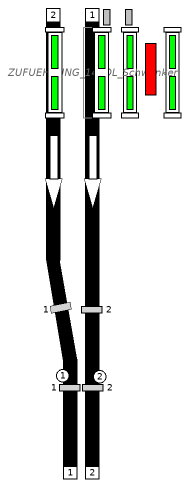
embedded screen at (73,127)-(90,200): SIGNS_ARROWDOWN
rounded rectangle at (74,0)-(88,14): text "1"; alarm colour if ST03_562_B69_0.BitInToCheck; tooltip ST03_562_B69_0
rounded rectangle at (74,458)-(88,471): text "2"; alarm colour if ST03_563_B70_7.BitInToCheck; tooltip ST03_563_B70_7
ellipse at (82,362)-(95,375): text "2"; alarm colour if ST03_563_B70_6.BitInToCheck; tooltip ST03_563_B70_6
rectangle at (71,376)-(92,383): alarm colour if ST03_563_B70_4.ValveSensor; tooltip ST03_563_B70_3
rectangle at (36,373)-(49,386): text "1"
rectangle at (92,373)-(105,386): text "2"
embedded screen at (110,19)-(170,110): ZUFUEHRUNG_268POL_RP_SCHWENKER; invisible if NOT ST03_564_Y71_5.SensorInitIn[1].SensorSignal
rectangle at (114,1)-(121,17): alarm colour if ST03_564_Y71_5.SensorInitIn[1].SensorSignal; tooltip ST03_564_Y71_5.SensorInitIn[1].SensorSignal
rectangle at (92,1)-(99,17): alarm colour if ST03_564_Y71_5.SensorWorkIn[1].SensorSignal; tooltip ST03_564_Y71_5.SensorWorkIn[1].SensorSignal
embedded screen at (72,19)-(91,110): ZUFUEHRUNG_14POL_Schwenker; invisible if NOT ST03_512_B69_6.ValveSensor
rectangle at (48,376)-(69,383): alarm colour if ST03_562_B69_4.ValveSensor; tooltip ST03_564_Y71_1
rounded rectangle at (52,458)-(66,471): text "1"; alarm colour if ST03_562_B67_7.BitInToCheck; tooltip ST03_562_B67_7
ellipse at (45,361)-(58,374): text "1"; alarm colour if ST03_562_B69_6.BitInToCheck; tooltip ST03_562_B69_6
embedded screen at (34,19)-(100,110): ZUFUEHRUNG_268POL_RP_SCHWENKER; invisible if NOT ST03_564_Y71_5.SensorWorkIn[1].SensorSignal
embedded screen at (34,127)-(51,200): SIGNS_ARROWDOWN
rectangle at (70,298)-(91,305): alarm colour if ST03_563_B70_2.ValveSensor; tooltip ST03_564_Y71_2
rectangle at (28,295)-(41,308): text "1"
rectangle at (91,295)-(104,308): text "2"
polygon at (39,294)-(60,305): alarm colour if ST03_562_B69_2.ValveSensor; tooltip ST03_564_Y71_0
rounded rectangle at (134,35)-(145,87): alarm colour if ST03_Init_Lockings.b_freiFuerSG; tooltip b_freiFuerSG
rounded rectangle at (35,0)-(49,14): text "2"; alarm colour if ST03_563_B70_0.BitInToCheck; tooltip ST03_563_B70_0
5 more shapes without text or variables
*)

(* Visualisation ZUFUEHRUNG_268POL_RP_SCHWENKER
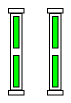
rectangle at (44,8)-(50,40): invisible if NOT $Reihe1$
rectangle at (44,47)-(50,79): invisible if NOT $Reihe1$
rounded rectangle at (39,0)-(55,5): invisible if NOT ST03_564_Y71_5.SensorWorkIn[1].SensorSignal; alarm colour if $Reihe1$; tooltip ST03_565_B72_0
rounded rectangle at (39,82)-(55,87): invisible if NOT ST03_564_Y71_5.SensorWorkIn[1].SensorSignal; alarm colour if $Reihe1$; tooltip ST03_565_B72_0
rectangle at (5,8)-(11,40): invisible if NOT $Reihe2$
rectangle at (5,47)-(11,79): invisible if NOT $Reihe2$
rounded rectangle at (0,0)-(16,5): invisible if NOT ST03_564_Y71_5.SensorWorkIn[1].SensorSignal; alarm colour if $Reihe2$; tooltip ST03_565_B72_1
rounded rectangle at (0,82)-(16,87): invisible if NOT ST03_564_Y71_5.SensorWorkIn[1].SensorSignal; alarm colour if $Reihe2$; tooltip ST03_565_B72_1
2 more shapes without text or variables
*)

(* Visualisation ZUFUEHRUNG_33POL
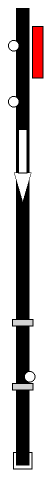
embedded screen at (9,126)-(26,199): SIGNS_ARROWDOWN
ellipse at (3,37)-(14,48): alarm colour if ST03_571_B69_0.BitInToCheck; tooltip ST03_501_B69_0
ellipse at (19,368)-(30,379): alarm colour if ST03_571_B69_6.BitInToCheck; tooltip ST03_501_B69_6
rectangle at (7,380)-(28,387): alarm colour if ST03_571_B69_5.ValveSensor; tooltip ST03_501_B69_3
rectangle at (7,316)-(28,323): alarm colour if ST03_571_B69_3.ValveSensor; tooltip ST03_501_B69_1
rounded rectangle at (8,449)-(27,466): alarm colour if ST03_571_B69_7.BitInToCheck; tooltip ST03_502_B70_0
rounded rectangle at (27,23)-(38,75): alarm colour if ST03_Init_Lockings.b_freiFuerSG; tooltip b_freiFuerSG
ellipse at (3,93)-(14,104): alarm colour if ST03_571_B69_1.BitInToCheck; tooltip ST03_501_B69_0
2 more shapes without text or variables
*)

(* Visualisation ZUFUEHRUNG_35POL
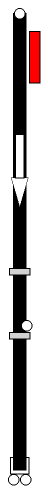
ellipse at (6,466)-(17,477): alarm colour if ST08_412_B58_6_35pol.BitInToCheck; tooltip ST08_412_B58_6_35pol
embedded screen at (9,126)-(26,199): SIGNS_ARROWDOWN
ellipse at (18,466)-(29,477): alarm colour if ST08_412_B58_5_35pol.BitInToCheck; tooltip ST08_412_B58_5_35pol
ellipse at (12,0)-(23,11): alarm colour if ST08_412_B58_4.BitInToCheck; tooltip ST08_412_B58_4
ellipse at (19,312)-(30,323): alarm colour if ST08_412_B58_7.BitInToCheck; tooltip ST08_412_B58_7
rectangle at (7,324)-(28,331): alarm colour if ST08_412_B58_2.ValveSensor; tooltip ST08_412_B58_2
rectangle at (7,260)-(28,267): alarm colour if ST08_412_B58_0.ValveSensor; tooltip ST08_412_B58_0
rounded rectangle at (8,449)-(27,466): alarm colour if ST08_412_B59_0.BitInToCheck; tooltip ST08_412_B59_0
rounded rectangle at (27,23)-(38,75): alarm colour if ST03_Init_Lockings.b_freiFuerSG; tooltip b_freiFuerSG
2 more shapes without text or variables
*)

(* Visualisation ZUFUEHRUNG_46POL
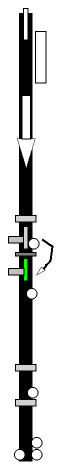
ellipse at (37,446)-(48,457): alarm colour if ST03_462_B70_1.BitInToCheck; tooltip ST03_462_B70_1
embedded screen at (23,92)-(41,165): SIGNS_ARROWDOWN
ellipse at (20,446)-(31,457): alarm colour if ST03_462_B70_2.BitInToCheck; tooltip ST03_462_B70_2
ellipse at (37,434)-(48,445): alarm colour if ST03_463_B70_7.BitInToCheck; tooltip ST03_463_B70_7
ellipse at (33,384)-(44,395): alarm colour if ST03_461_B69_7.BitInToCheck; tooltip ST03_461_B69_7
rectangle at (21,396)-(42,403): alarm colour if ST03_461_B69_2.ValveSensor; tooltip ST03_461_B69_2
rectangle at (21,361)-(42,368): alarm colour if ST03_461_B69_0.ValveSensor; tooltip ST03_461_B69_0
rounded rectangle at (41,28)-(52,80): alarm colour if ST03_Init_Lockings.b_freiFuerSG; tooltip b_freiFuerSG
rounded rectangle at (29,5)-(34,37): alarm colour if ST03_461_B69_4.BitInToCheck; tooltip ST03_461_B69_4
rectangle at (21,212)-(42,219): alarm colour if ST03_461_B69_5.ValveSensor; tooltip ST03_461_B69_5
rectangle at (14,233)-(30,240): invisible if NOT ST03_463_B70_5.ValveSensor; alarm colour if ST03_464_B71_6.BitInToCheck; tooltip ST03_464_B71_6; x offset ST03_CallFBs.ST03_463_B70_3_4_pos
rectangle at (29,223)-(34,246): invisible if NOT ST03_463_B70_5.ValveSensor; alarm colour if ST03_462_B70_0.BitInToCheck
rectangle at (29,255)-(34,278): invisible if NOT ST03_463_B70_6.ValveSensor
rectangle at (14,265)-(30,272): invisible if NOT ST03_463_B70_6.ValveSensor; alarm colour if ST03_464_B71_6.BitInToCheck; tooltip ST03_464_B71_6; x offset ST03_CallFBs.ST03_463_B70_3_4_pos
ellipse at (32,285)-(43,296): alarm colour if ST03_464_B71_7.BitInToCheck; tooltip ST03_464_B71_7
curve at (48,236)-(58,266): invisible if NOT ST03_463_B70_5.ValveSensor AND NOT NOT ST03_463_B70_5.ValveSensor
polygon at (42,264)-(51,272): invisible if NOT ST03_463_B70_5.ValveSensor AND NOT NOT ST03_463_B70_5.ValveSensor
ellipse at (34,235)-(45,246): alarm colour if ST03_462_B70_0.BitInToCheck; tooltip ST03_462_B70_0
2 more shapes without text or variables
*)

(* Visualisation ZUFUEHRUNG_48POL
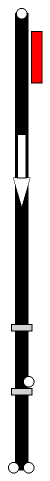
embedded screen at (9,126)-(26,199): SIGNS_ARROWDOWN
ellipse at (12,0)-(23,11): alarm colour if ST03_551_B69_0.BitInToCheck; tooltip ST03_541_B69_0
ellipse at (19,368)-(30,379): alarm colour if ST03_551_B69_6.BitInToCheck; tooltip ST03_541_B69_6
rectangle at (7,380)-(28,387): alarm colour if ST03_551_B69_4.ValveSensor; tooltip ST03_541_B69_3
rectangle at (7,316)-(28,323): alarm colour if ST03_551_B69_2.ValveSensor; tooltip ST03_541_B69_1
rounded rectangle at (27,23)-(38,75): alarm colour if ST03_Init_Lockings.b_freiFuerSG; tooltip b_freiFuerSG
ellipse at (4,454)-(15,465): alarm colour if ST03_552_B70_0.BitInToCheck; tooltip ST03_542_B70_0
ellipse at (19,454)-(30,465): alarm colour if ST03_551_B69_7.BitInToCheck; tooltip ST03_542_B70_0
2 more shapes without text or variables
*)

(* Visualisation ZUFUEHRUNG_72POL
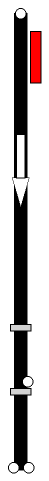
embedded screen at (9,126)-(26,199): SIGNS_ARROWDOWN
ellipse at (12,0)-(23,11): alarm colour if ST03_546_B69_0.BitInToCheck; tooltip ST03_541_B69_0
ellipse at (19,368)-(30,379): alarm colour if ST03_546_B69_6.BitInToCheck; tooltip ST03_541_B69_6
rectangle at (7,380)-(28,387): alarm colour if ST03_546_B69_4.ValveSensor; tooltip ST03_541_B69_3
rectangle at (7,316)-(28,323): alarm colour if ST03_546_B69_2.ValveSensor; tooltip ST03_541_B69_1
rounded rectangle at (27,23)-(38,75): alarm colour if ST03_Init_Lockings.b_freiFuerSG; tooltip b_freiFuerSG
ellipse at (5,454)-(16,465): alarm colour if ST03_547_B70_0.BitInToCheck; tooltip ST03_542_B70_0
ellipse at (20,454)-(31,465): alarm colour if ST03_546_B69_7.BitInToCheck; tooltip ST03_542_B70_0
2 more shapes without text or variables
*)

(* Visualisation ZUFUEHRUNG_74_91_168POL
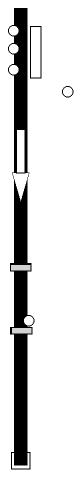
rounded rectangle at (8,444)-(27,461): invisible if NOT MP.ST03.SGM_3621; alarm colour if ST03_422_B64_4.BitInToCheck
ellipse at (5,35)-(16,46): invisible if MP.ST03.SGM_3621; alarm colour if ST08_412_B58_5.BitInToCheck
embedded screen at (9,121)-(26,194): SIGNS_ARROWDOWN
ellipse at (5,56)-(16,67): invisible if MP.ST03.SGM_3621 OR gTypeCode=379; alarm colour if ST08_412_B58_6.BitInToCheck
ellipse at (5,17)-(16,28): invisible if MP.ST03.SGM_3621; alarm colour if ST08_412_B58_4.BitInToCheck
ellipse at (19,307)-(30,318): invisible if MP.ST03.SGM_3621; alarm colour if ST08_412_B58_7.BitInToCheck
rectangle at (7,319)-(28,326): invisible if MP.ST03.SGM_3621; alarm colour if ST08_412_B58_2.ValveSensor
rectangle at (7,255)-(28,262): invisible if MP.ST03.SGM_3621; alarm colour if ST08_412_B58_0.ValveSensor
rounded rectangle at (8,444)-(27,461): invisible if MP.ST03.SGM_3621; alarm colour if ST08_412_B59_0.BitInToCheck; tooltip ST08_412_B59_0
rounded rectangle at (27,18)-(38,70): alarm colour if ST03_Init_Lockings.b_freiFuerSG; tooltip b_freiFuerSG
rectangle at (8,319)-(29,326): invisible if NOT MP.ST03.SGM_3621; alarm colour if ST03_421_B63_2.ValveSensor; tooltip ST03_421_B63_2
ellipse at (5,35)-(16,46): invisible if NOT MP.ST03.SGM_3621; alarm colour if ST03_421_B63_5.BitInToCheck; tooltip ST03_421_B63_5
ellipse at (59,78)-(70,89): invisible if NOT MP.ST03.SGM_3621; alarm colour if ST03_421_B63_6.BitInToCheck; tooltip ST03_421_B63_6
ellipse at (5,17)-(16,28): invisible if NOT MP.ST03.SGM_3621; alarm colour if ST03_421_B63_4.BitInToCheck; tooltip ST03_421_B63_4
rectangle at (7,256)-(28,263): invisible if NOT MP.ST03.SGM_3621; alarm colour if ST03_421_B63_0.ValveSensor; tooltip ST03_421_B63_0
ellipse at (20,307)-(31,318): invisible if NOT MP.ST03.SGM_3621; alarm colour if ST03_421_B63_7.BitInToCheck; tooltip ST03_421_B63_7
2 more shapes without text or variables
*)

(* Visualisation ZUFUEHRUNG_7POL
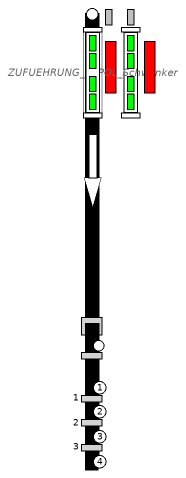
embedded screen at (16,126)-(33,199): SIGNS_ARROWDOWN
ellipse at (18,0)-(30,12): alarm colour if ST03_514_B71_7.BitInToCheck; tooltip ST03_514_B71_7
ellipse at (25,332)-(36,343): alarm colour if ST03_513_B70_4.BitInToCheck; tooltip ST03_513_B70_4
rectangle at (13,344)-(34,351): alarm colour if ST03_513_B70_3. ValveSensor; tooltip ST03_513_B70_3
rectangle at (13,309)-(34,327): alarm colour if ST03_513_B70_0.ValveSensor; tooltip ST03_513_B70_0
rounded rectangle at (37,33)-(48,85): alarm colour if ST03_Init_Lockings.b_freiFuerSG; tooltip b_freiFuerSG
ellipse at (25,447)-(38,460): text "4"; alarm colour if ST03_514_B71_6.BitInToCheck; tooltip ST03_514_B71_6
ellipse at (25,422)-(38,435): text "3"; alarm colour if ST03_514_B71_5.BitInToCheck; tooltip ST03_514_B71_5
rectangle at (13,436)-(34,443): alarm colour if ST03_514_B71_4.ValveSensor; tooltip ST03_514_B71_4
ellipse at (25,397)-(38,410): text "2"; alarm colour if ST03_514_B71_2.BitInToCheck; tooltip ST03_514_B71_2
rectangle at (13,411)-(34,418): alarm colour if ST03_514_B71_1.ValveSensor; tooltip ST03_514_B71_1
ellipse at (25,373)-(38,386): text "1"; alarm colour if ST03_513_B70_7.BitInToCheck; tooltip ST03_513_B70_7
rectangle at (13,387)-(34,394): alarm colour if ST03_513_B70_6.ValveSensor; tooltip ST03_513_B70_6
rectangle at (1,383)-(14,396): text "1"
rectangle at (1,408)-(14,421): text "2"
rectangle at (1,432)-(14,445): text "3"
embedded screen at (53,19)-(72,110): ZUFUEHRUNG_7POL_Schwenker; invisible if NOT ST03_515_Y72_1.SensorInitIn[1].SensorSignal
rectangle at (59,1)-(66,17): alarm colour if ST03_515_Y72_1.SensorInitIn[1].SensorSignal; tooltip ST03_515_Y72_1
rectangle at (37,1)-(44,17): alarm colour if ST03_515_Y72_1.SensorWorkIn[1].SensorSignal; tooltip ST03_515_Y72_1
embedded screen at (15,19)-(34,110): ZUFUEHRUNG_14POL_Schwenker; invisible if NOT ST03_512_B69_6.ValveSensor
embedded screen at (15,19)-(34,110): ZUFUEHRUNG_7POL_Schwenker; invisible if NOT ST03_515_Y72_1.SensorWorkIn[1].SensorSignal
rounded rectangle at (76,33)-(87,85): alarm colour if ST00_73_K4.BitInToCheck; tooltip ST00_73_K4
3 more shapes without text or variables
*)

(* Visualisation ZUFUEHRUNG_7POL_SCHWENKER
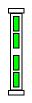
rectangle at (5,8)-(11,23): invisible if NOT ST03_512_XG1.BitInToCheck
rectangle at (5,25)-(11,40): invisible if NOT ST03_512_XG1.BitInToCheck
rectangle at (5,47)-(11,62): invisible if NOT ST03_512_XG1.BitInToCheck
rectangle at (5,64)-(11,79): invisible if NOT ST03_512_XG1.BitInToCheck
rounded rectangle at (0,0)-(16,5): invisible if ST03_515_Y72_1.SensorWorkIn[1].SensorSignal; alarm colour if ST03_512_XG1.BitInToCheck
rounded rectangle at (0,82)-(16,87): invisible if ST03_515_Y72_1.SensorWorkIn[1].SensorSignal; alarm colour if ST03_512_XG1.BitInToCheck
1 more shapes without text or variables
*)

(* Visualisation ZUFUEHRUNG_88POL
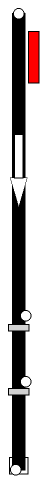
embedded screen at (9,126)-(26,199): SIGNS_ARROWDOWN
ellipse at (12,0)-(23,11): alarm colour if ST03_501_B69_0.BitInToCheck; tooltip ST03_501_B69_0
ellipse at (19,368)-(30,379): alarm colour if ST03_501_B69_6.BitInToCheck; tooltip ST03_501_B69_6
rectangle at (7,380)-(28,387): alarm colour if ST03_501_B69_3.ValveSensor; tooltip ST03_501_B69_3
rectangle at (7,316)-(28,323): alarm colour if ST03_501_B69_1.ValveSensor; tooltip ST03_501_B69_1
rounded rectangle at (8,449)-(27,466): alarm colour if ST03_502_B70_0.BitInToCheck; tooltip ST03_502_B70_0
rounded rectangle at (27,23)-(38,75): alarm colour if ST03_Init_Lockings.b_freiFuerSG; tooltip b_freiFuerSG
ellipse at (19,302)-(30,313): alarm colour if ST03_501_B69_5.BitInToCheck; tooltip ST03_501_B69_5
ellipse at (9,456)-(20,467): alarm colour if ST03_501_B69_7.BitInToCheck; tooltip ST03_501_B69_7
2 more shapes without text or variables
*)

(* Visualisation ZUFUEHRUNG_88POL_AMG
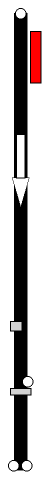
embedded screen at (9,126)-(26,199): SIGNS_ARROWDOWN
ellipse at (12,0)-(23,11): alarm colour if ST03_521_B69_0.BitInToCheck; tooltip ST03_521_B69_0
ellipse at (19,368)-(30,379): alarm colour if ST03_521_B69_6.BitInToCheck; tooltip ST03_521_B69_6
rectangle at (7,380)-(28,387): alarm colour if ST03_521_B69_4.ValveSensor; tooltip ST03_521_B69_3
rectangle at (7,313)-(19,323): alarm colour if ST03_521_B69_2.ValveSensor; tooltip ST03_521_B69_1
rounded rectangle at (27,23)-(38,75): alarm colour if ST03_Init_Lockings.b_freiFuerSG; tooltip b_freiFuerSG
ellipse at (5,452)-(16,463): alarm colour if ST03_521_B69_7.BitInToCheck; tooltip ST03_521_B69_7
ellipse at (18,452)-(29,463): alarm colour if ST03_522_B70_0.BitInToCheck; tooltip ST03_522_B70_0
2 more shapes without text or variables
*)

(* Visualisation ZUFUEHRUNG_92POL
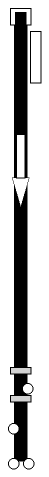
ellipse at (30,455)-(41,466): alarm colour if ST03_445_B70_1.BitInToCheck; tooltip ST03_445_B70_1
embedded screen at (19,131)-(36,204): SIGNS_ARROWDOWN
ellipse at (15,455)-(26,466): alarm colour if ST03_445_B70_2.BitInToCheck; tooltip ST03_445_B70_2
ellipse at (15,420)-(26,431): alarm colour if ST03_446_B70_4.BitInToCheck; tooltip ST03_446_B70_4
ellipse at (29,380)-(40,391): alarm colour if ST03_444_B69_7.BitInToCheck; tooltip ST03_444_B69_7
rectangle at (17,392)-(38,399): alarm colour if ST03_444_B69_2.ValveSensor; tooltip ST03_444_B69_2
rectangle at (17,364)-(38,371): alarm colour if ST03_444_B69_0.ValveSensor; tooltip ST03_444_B69_0
rounded rectangle at (17,5)-(38,22): alarm colour if ST03_435_B67_4.BitInToCheck; tooltip ST03_435_B67_4
rounded rectangle at (37,28)-(48,80): alarm colour if ST03_Init_Lockings.b_freiFuerSG; tooltip b_freiFuerSG
2 more shapes without text or variables
*)

(* Visualisation ZUFUEHRUNG_93POL
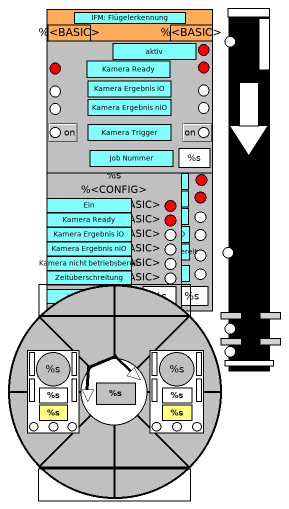
embedded screen at (40,160)-(206,303): ZLIB_SENSOPART_1; invisible if gTypeCode<>4991 AND gTypeCode <>312 OR MP.ST02.SensopartEthernet
embedded screen at (40,160)-(175,303): ZLIB_SENSOPART_5; invisible if gTypeCode<>4991 AND gTypeCode <>312 OR NOT MP.ST02.SensopartEthernet
embedded screen at (0,276)-(215,493): ROUNDTABLE; invisible if gTypeCode<>4991 AND gTypeCode <>312
embedded screen at (40,1)-(206,165): ZLIB_IFM; invisible if gTypeCode<>4991 AND gTypeCode <>312
ellipse at (218,28)-(229,39): alarm colour if NOT ST02_FDB_40_B61.BitInToCheck; tooltip ST02_FDB_40_B61
embedded screen at (223,74)-(261,147): SIGNS_ARROWDOWN
ellipse at (218,315)-(229,326): alarm colour if ST00_72_X1_3.BitInToCheck; tooltip ST00_72_X1_3
rectangle at (214,304)-(235,311): alarm colour if ST00_74_Y2_5.SensorWorkIn[1].SensorSignal; tooltip ST00_74_Y2_5
rectangle at (253,304)-(274,311): alarm colour if ST00_74_Y2_5.SensorWorkIn[2].SensorSignal; tooltip ST00_74_Y2_5
rectangle at (214,330)-(235,337): alarm colour if NOT ST00_74_Y2_4.SensorWorkIn[1].SensorSignal; tooltip ST00_74_Y2_4
rectangle at (253,330)-(274,337): alarm colour if NOT ST00_74_Y2_4.SensorWorkIn[2].SensorSignal; tooltip ST00_74_Y2_4
rectangle at (222,342)-(263,363): invisible if gTypeCode<>4991
ellipse at (218,338)-(229,349): invisible if gTypeCode<>4991; alarm colour if ST02_FDB_80_B02.BitInToCheck; tooltip ST02_FDB_80_B02
rectangle at (218,352)-(267,358): invisible if gTypeCode<>4991
ellipse at (216,239)-(227,250): alarm colour if NOT ST02_FDB_40_B71.BitInToCheck; tooltip ST02_FDB_40_B71
rectangle at (225,149)-(259,156): alarm colour if ST02_FDB_54_B41.BitInToCheck
rounded rectangle at (252,10)-(263,62): alarm colour if ST03_Init_Lockings.b_freiFuerSG; tooltip b_freiFuerSG
rounded rectangle at (221,0)-(263,9): alarm colour if ST02_S1_40K01.BitInToCheck; tooltip ST02_S1_40K01
rectangle at (222,194)-(262,200): alarm colour if ST02_FDB_54_B21.ValveSensor
1 more shapes without text or variables
*)

(* Visualisation ZUFUEHRUNG_NOX_4POL
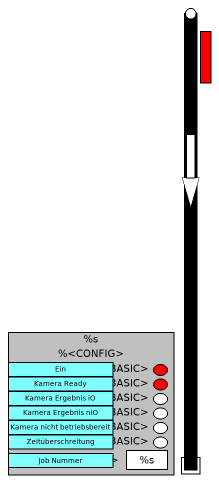
embedded screen at (174,126)-(191,199): SIGNS_ARROWDOWN
ellipse at (177,0)-(188,11): alarm colour if ST03_491_B69_0.BitInToCheck; tooltip ST03_491_B69_0
ellipse at (6,394)-(17,405): alarm colour if ST03_491_B69_5.BitInToCheck; tooltip ST03_491_B69_5
rectangle at (7,406)-(28,413): alarm colour if ST03_491_B69_2.ValveSensor; tooltip ST03_491_B69_2
rectangle at (7,371)-(28,378): alarm colour if ST03_491_B69_1.ValveSensor; tooltip ST03_491_B69_1
rounded rectangle at (173,449)-(192,466): alarm colour if ST03_491_B69_7.BitInToCheck; tooltip ST03_491_B69_7
rounded rectangle at (192,23)-(203,75): alarm colour if ST03_Init_Lockings.b_freiFuerSG; tooltip b_freiFuerSG
embedded screen at (0,324)-(166,467): ZLIB_SENSOPART_5; invisible if TRUE
2 more shapes without text or variables
*)

(* Visualisation ZUFUEHRUNG_NOX_5_6POL
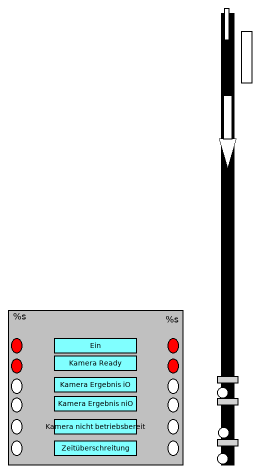
embedded screen at (274,87)-(291,160): SIGNS_ARROWDOWN
ellipse at (272,445)-(283,456): alarm colour if ST03_4x3_B70_1.BitInToCheck; tooltip ST03_4x3_B70_1
ellipse at (273,419)-(284,430): alarm colour if ST03_4x3_B70_0.BitInToCheck; tooltip ST03_4x3_B70_0
rectangle at (272,431)-(293,438): alarm colour if ST03_4x2_B69_7.ValveSensor; tooltip ST03_4x2_B69_7
rectangle at (272,390)-(293,397): alarm colour if ST03_4x2_B69_4.ValveSensor; tooltip ST03_4x2_B69_4
rounded rectangle at (296,23)-(307,75): alarm colour if ST03_Init_Lockings.b_freiFuerSG; tooltip b_freiFuerSG
rounded rectangle at (279,0)-(284,32): alarm colour if ST03_4x2_B69_0.BitInToCheck; tooltip ST03_4x2_B69_0
rounded rectangle at (272,368)-(293,375): alarm colour if ST03_4x2_B69_2.ValveSensor; tooltip ST03_4x2_B69_2
ellipse at (272,379)-(283,390): alarm colour if ST03_4x2_B69_5.BitInToCheck; tooltip ST03_4x2_B69_5
embedded screen at (63,302)-(238,457): ZLIB_SENSOPART_6; invisible if gTypeCode <> 4993
1 more shapes without text or variables
*)

(* Visualisation DOOR_LOCK
rectangle at (0,0)-(31,31): invisible if $lock$ AND NOT $visibal_open$; alarm colour if NOT $lock$
rectangle at (0,0)-(31,31): invisible if NOT $open$
*)

(* Visualisation MIN_EXIT
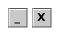
button at (1,0)-(20,19): text "_"; shows 'ST_MinExit.btn_min.Text'; invisible if ST_MinExit.btn_min.Visible; taps ST_MinExit.btn_min.Pressed; dynamic style ST_MinExit.btn_min.TextColor, ST_MinExit.btn_min.BackgroundColor, ST_MinExit.btn_min.BackgroundColor, ST_MinExit.btn_min.Enable
button at (25,0)-(44,19): text "X"; shows 'ST_MinExit.btn_exit.Text'; invisible if ST_MinExit.btn_exit.Visible; taps ST_MinExit.btn_exit.Pressed; runs INTERN EXITPROGRAM; dynamic style ST_MinExit.btn_exit.TextColor, ST_MinExit.btn_exit.BackgroundColor, ST_MinExit.btn_exit.BackgroundColor, ST_MinExit.btn_exit.Enable
*)

(* Visualisation SPRACHE_MENUE
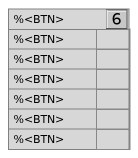
rectangle at (0,20)-(121,41): text "%<BTN>"; shows ST_Lng.btn_Language[0].Text; invisible if NOT ST_Lng.fb_ton_ausblenden.IN OR ST_Lng.btn_Language[0].unsichtbar; taps ST_Lng.btn_Language[0].tasten; runs INTERN LANGUAGE DE; dynamic style Visu.System.btn_Language[0].TextFarbe, ST_Lng.btn_Language[0].deaktivieren
rectangle at (0,40)-(121,61): text "%<BTN>"; shows ST_Lng.btn_Language[1].Text; invisible if NOT ST_Lng.fb_ton_ausblenden.IN OR ST_Lng.btn_Language[1].unsichtbar; taps ST_Lng.btn_Language[1].tasten; runs INTERN LANGUAGE EN; dynamic style Visu.System.btn_Language[1].TextFarbe, ST_Lng.btn_Language[1].deaktivieren
rectangle at (0,60)-(121,81): text "%<BTN>"; shows ST_Lng.btn_Language[2].Text; invisible if NOT ST_Lng.fb_ton_ausblenden.IN OR ST_Lng.btn_Language[2].unsichtbar; taps ST_Lng.btn_Language[2].tasten; runs INTERN LANGUAGE CZ; dynamic style Visu.System.btn_Language[2].TextFarbe, ST_Lng.btn_Language[2].deaktivieren
rectangle at (0,80)-(121,101): text "%<BTN>"; shows ST_Lng.btn_Language[3].Text; invisible if NOT ST_Lng.fb_ton_ausblenden.IN OR ST_Lng.btn_Language[3].unsichtbar; taps ST_Lng.btn_Language[3].tasten; runs INTERN LANGUAGE; dynamic style Visu.System.btn_Language[3].TextFarbe, ST_Lng.btn_Language[3].deaktivieren
rectangle at (0,100)-(121,121): text "%<BTN>"; shows ST_Lng.btn_Language[4].Text; invisible if NOT ST_Lng.fb_ton_ausblenden.IN OR ST_Lng.btn_Language[4].unsichtbar; taps ST_Lng.btn_Language[4].tasten; runs INTERN LANGUAGE; dynamic style Visu.System.btn_Language[4].TextFarbe, ST_Lng.btn_Language[4].deaktivieren
rectangle at (0,120)-(121,141): text "%<BTN>"; shows ST_Lng.btn_Language[5].Text; invisible if NOT ST_Lng.fb_ton_ausblenden.IN OR ST_Lng.btn_Language[5].unsichtbar; taps ST_Lng.btn_Language[5].tasten; runs INTERN LANGUAGE; dynamic style Visu.System.btn_Language[5].TextFarbe, ST_Lng.btn_Language[5].deaktivieren
other_BMP at (88,20)-(122,41): invisible if NOT ST_Lng.fb_ton_ausblenden.IN OR ST_Lng.btn_Language[0].unsichtbar; taps ST_Lng.btn_Language[0].tasten; dynamic style ST_Lng.btn_Language[0].BmpPath
other_BMP at (88,40)-(122,61): invisible if NOT ST_Lng.fb_ton_ausblenden.IN OR ST_Lng.btn_Language[1].unsichtbar; taps ST_Lng.btn_Language[1].tasten; dynamic style ST_Lng.btn_Language[1].BmpPath
other_BMP at (88,60)-(122,81): invisible if NOT ST_Lng.fb_ton_ausblenden.IN OR ST_Lng.btn_Language[2].unsichtbar; taps ST_Lng.btn_Language[2].tasten; dynamic style ST_Lng.btn_Language[2].BmpPath
other_BMP at (88,80)-(122,101): invisible if NOT ST_Lng.fb_ton_ausblenden.IN OR ST_Lng.btn_Language[3].unsichtbar; taps ST_Lng.btn_Language[3].tasten; dynamic style ST_Lng.btn_Language[3].BmpPath
other_BMP at (88,100)-(122,121): invisible if NOT ST_Lng.fb_ton_ausblenden.IN OR ST_Lng.btn_Language[4].unsichtbar; taps ST_Lng.btn_Language[4].tasten; dynamic style ST_Lng.btn_Language[4].BmpPath
other_BMP at (88,120)-(122,141): invisible if NOT ST_Lng.fb_ton_ausblenden.IN OR ST_Lng.btn_Language[5].unsichtbar; taps ST_Lng.btn_Language[5].tasten; dynamic style ST_Lng.btn_Language[5].BmpPath
rectangle at (0,0)-(121,21): text "%<BTN>"; shows ST_Lng.btn_Language[ST_Lng.index].Text; invisible if ST_Lng.btn_Language[ST_Lng.index].unsichtbar; taps ST_Lng.b_einblenden; dynamic style Visu.System.btn_Language[ST_System.index].TextFarbe, ST_Lng.btn_Language[ST_System.index].innenFarbe, ST_Lng.btn_Language[ST_Lng.index].deaktivieren
button at (98,1)-(119,20): text "6"; shows '0xEA'; taps ST_Lng.b_einblenden; dynamic style Color.lightgrey, Color.lightgrey
*)

(* Visualisation TEILEZAEHLER
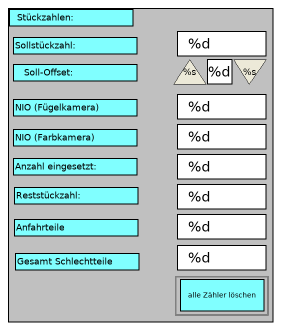
rectangle at (0,0)-(265,314): text "%<DATA>"; shows 'Parts'
rectangle at (10,23)-(157,48): text "%<DATA>"; shows 'PartsToProduce'
rectangle at (169,23)-(258,48): text "%d"; shows MP.ST00.PartsToProduce; editable 0..
rectangle at (10,51)-(157,76): text "%<DATA>"; shows 'PartsToProduceOffset'
rectangle at (199,51)-(224,76): text "%d"; shows MP.ST00.PartsToProduceOffset; editable 0..
rectangle at (10,146)-(157,171): text "%<DATA>"; shows 'gPartsInserted'
rectangle at (169,146)-(258,171): text "%d"; shows gPartsInserted; editable 0..
rectangle at (10,176)-(157,201): text "%<DATA>"; shows 'PartsRemaining'
rectangle at (169,176)-(258,201): text "%d"; shows MP.ST00.PartsRemaining; editable
embedded screen at (165,51)-(198,76): ZLIB_VISUBUTTON_ARROW_UP
embedded screen at (225,51)-(258,76): ZLIB_VISUBUTTON_ARROW_DOWN
embedded screen at (167,268)-(260,307): ZLIB_VISUBUTTON_S18
rectangle at (10,116)-(157,141): text "%<DATA>"; shows 'gNokPartsColorCam'; invisible if gTypeCode<>5633 AND gTypeCode<>4991 AND gTypeCode <>312 AND gTypeCode <>322
rectangle at (10,86)-(157,111): text "%<DATA>"; shows 'gNokPartsWingCam'; invisible if gTypeCode<>4991 AND gTypeCode <>312
rectangle at (169,86)-(258,111): text "%d"; shows gNokPartsWingCam; invisible if gTypeCode<>4991 AND gTypeCode <>312; editable 0..
rectangle at (169,116)-(258,141): text "%d"; shows gNokPartsColorCam; invisible if gTypeCode<>5633 AND gTypeCode<>4991 AND gTypeCode <>312 AND gTypeCode <>322; editable 0..
rectangle at (1,1)-(125,18): text "Stückzahlen:"; invisible if TRUE
rectangle at (5,29)-(129,46): text "Sollstückzahl:"; invisible if TRUE
rectangle at (5,56)-(129,73): text "Soll-Offset:"; invisible if TRUE
rectangle at (5,91)-(129,108): text "NIO (Fügelkamera)"; invisible if TRUE
rectangle at (5,121)-(129,138): text "NIO (Farbkamera)"; invisible if TRUE
rectangle at (5,150)-(129,167): text "Anzahl eingesetzt:"; invisible if TRUE
rectangle at (6,179)-(130,196): text "Reststückzahl:"; invisible if TRUE
rectangle at (172,271)-(256,303): text "alle Zähler löschen"; invisible if TRUE; dynamic style Color.lightgrey, Color.grey
rectangle at (10,207)-(166,232): text "%<DATA>"; shows 'Anfahrteile'
rectangle at (10,238)-(170,263): text "%<DATA>"; shows 'Gesamt Schlechtteile'
rectangle at (6,211)-(130,228): text "Anfahrteile"; invisible if TRUE
rectangle at (7,245)-(131,262): text "Gesamt Schlechtteile"; invisible if TRUE
rectangle at (169,206)-(258,231): text "%d"; shows i32_first_parts; editable 0..
rectangle at (169,237)-(258,262): text "%d"; shows i32_total_nok_parts; editable 0..
*)

(* Visualisation ZLIB_IFM
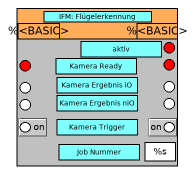
rectangle at (15,110)-(146,129): text "%<BASIC>"; shows 'Kamera Trigger'
rectangle at (15,69)-(146,88): text "%<BASIC>"; shows 'Kamera Ergebnis iO'
rectangle at (15,86)-(146,105): text "%<BASIC>"; shows 'Kamera Ergebnis niO'
ellipse at (147,73)-(158,84): alarm colour if ST02_FDB_56X1_6_IO.BitInToCheck
ellipse at (147,90)-(158,101): alarm colour if ST02_FDB_56X1_6_NIO.BitInToCheck
rectangle at (15,47)-(146,66): text "%<BASIC>"; shows 'Kamera Ready'
ellipse at (147,51)-(158,62): alarm colour if ST02_FDB_56X1_5_READY.BitInToCheck
rectangle at (40,134)-(121,153): text "%<BASIC>"; shows 'Job Nummer'
rectangle at (128,134)-(159,153): text "%s"; shows TD.IFM_CamProgNo; editable 0..3
ellipse at (147,34)-(158,45): alarm colour if MP.ST00.IFMCameraActive
ellipse at (3,74)-(14,85): alarm colour if ST02_FDB_55X1_6_IO.BitInToCheck
ellipse at (3,91)-(14,102): alarm colour if ST02_FDB_55X1_6_NIO.BitInToCheck
ellipse at (3,52)-(14,63): alarm colour if ST02_FDB_55X1_5_READY.BitInToCheck
rectangle at (62,30)-(143,49): text "%<BASIC>"; shows 'aktiv'
rectangle at (0,0)-(161,31): text "%<BASIC>"; shows 'IFM_Flügelerkennung'
rectangle at (1,15)-(43,31): text "%<BASIC>"; shows 'links'
button at (132,110)-(160,128): text "on"; invisible if ModeSelect.Mode <> 10; taps .ST02_FDB_56X1_2_TRIGGER.BitOutToSet; dynamic style color.lightgrey
ellipse at (147,114)-(158,124): alarm colour if .ST02_FDB_56X1_2_TRIGGER.BitOutToSet; taps .ST02_FDB_56X1_2_TRIGGER.BitOutToSet; dynamic style ModeSelect.Mode <> 10
button at (2,110)-(30,128): text "on"; invisible if ModeSelect.Mode <> 10; taps .ST02_FDB_55X1_2_TRIGGER.BitOutToSet; dynamic style color.lightgrey
ellipse at (3,114)-(14,124): alarm colour if .ST02_FDB_55X1_2_TRIGGER.BitOutToSet; taps .ST02_FDB_55X1_2_TRIGGER.BitOutToSet; dynamic style ModeSelect.Mode <> 10
rectangle at (64,33)-(145,49): text "aktiv"; invisible if TRUE
rectangle at (39,50)-(120,66): text "Kamera Ready"; invisible if TRUE
rectangle at (40,69)-(121,85): text "Kamera Ergebnis iO"; invisible if TRUE
rectangle at (40,87)-(121,103): text "Kamera Ergebnis niO"; invisible if TRUE
rectangle at (40,111)-(121,127): text "Kamera Trigger"; invisible if TRUE
rectangle at (42,136)-(123,152): text "Job Nummer"; invisible if TRUE
rectangle at (120,15)-(161,31): text "%<BASIC>"; shows 'rechts'
rectangle at (27,3)-(135,14): text "IFM: Flügelerkennung"; invisible if TRUE
1 more shapes without text or variables
*)

(* Visualisation ZLIB_OVERRIDE
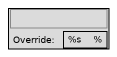
rectangle at (0,0)-(101,41): alarm colour if $override$<$overrideVorgabe$
other_SCROLLBAR at (2,1)-(99,20): top $override$; right 0; bottom 100
rounded rectangle at (0,23)-(57,41): text "Override:"; shows $override$; editable 0..100
rectangle at (55,23)-(99,40): text "%"; alarm colour if $override$<$overrideVorgabe$
rectangle at (55,23)-(99,40): text "%s"; shows $override$; editable 0..100
*)

(* Visualisation ZLIB_SCHWENKARM
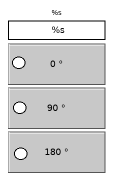
rectangle at (0,0)-(101,171): text "%s"; shows '$FB$'
rectangle at (2,13)-(99,32): text "%s"; shows $FB$.fb_state_entry.i16_step; alarm colour if $FB$.fb_state_entry.i16_step=1000
button at (2,36)-(99,77): text "0 °"; dynamic style Color.grey, TRUE
button at (2,80)-(99,121): text "90 °"; dynamic style Color.grey, TRUE
button at (2,124)-(99,165): text "180 °"; dynamic style Color.grey, TRUE
button at (2,36)-(99,77): text "0 °"; invisible if ModeSelect.Mode<>10; taps $FB$.b_0_grad; dynamic style color.lightgrey, Color.grey, ModeSelect.Mode<>10
button at (2,80)-(99,121): text "90 °"; invisible if ModeSelect.Mode<>10; taps $FB$.b_90_grad; dynamic style color.lightgrey, Color.grey, ModeSelect.Mode<>10
button at (2,124)-(99,165): text "180 °"; invisible if ModeSelect.Mode<>10; taps $FB$.b_180_grad; dynamic style color.lightgrey, Color.grey, ModeSelect.Mode<>10
ellipse at (6,49)-(19,61): alarm colour if $FB$.ST02_90_0_sens
ellipse at (7,94)-(20,106): alarm colour if $FB$.ST02_90_sens
ellipse at (8,140)-(21,152): alarm colour if $FB$.ST02_90_180_sens
*)

(* Visualisation ZLIB_ERRORHANDLER
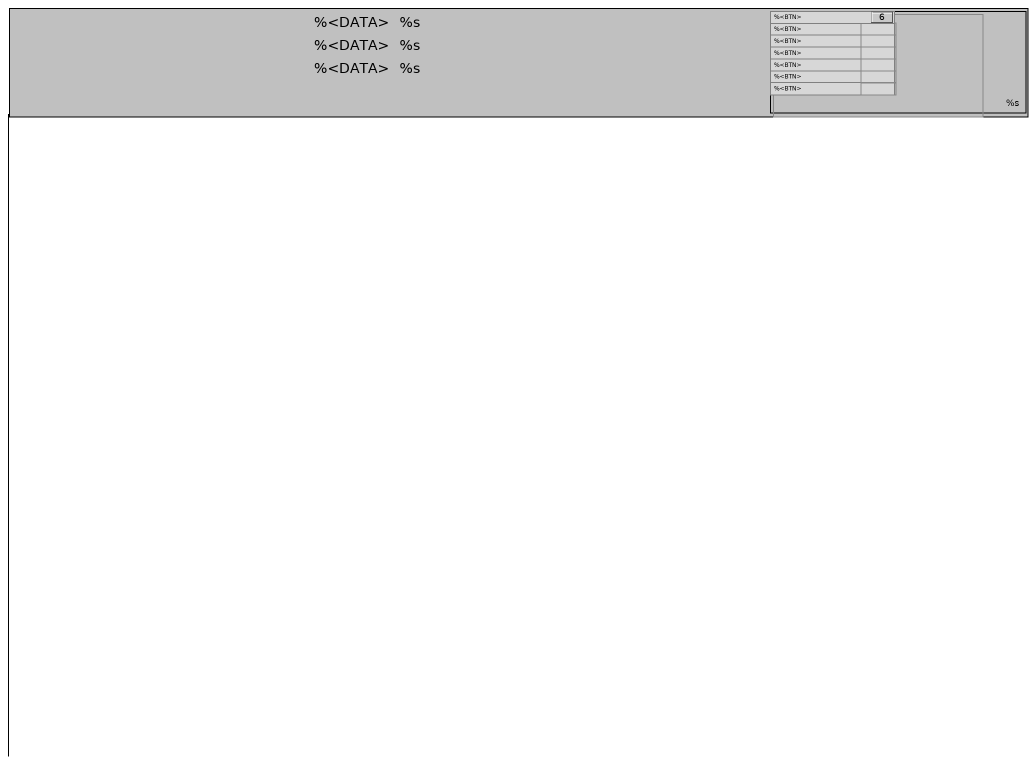
embedded screen at (0,106)-(1017,748): zLib_ErrorList
rectangle at (1,108)-(1020,759): opens ZOOMTOCALLER
rectangle at (886,87)-(1016,103): text "%s"; shows .gVarStrSystemTime
rectangle at (385,27)-(670,47): text "%s"; shows .TD.ArtNo
rectangle at (244,27)-(383,47): text "%<DATA>"; shows 'ArtNo'
rectangle at (385,4)-(670,24): text "%s"; shows .TD.TypeName
rectangle at (244,4)-(383,24): text "%<DATA>"; shows 'TypeName'
rectangle at (385,50)-(670,70): text "%s"; shows .TD.TypeDescription
rectangle at (244,50)-(383,70): text "%<DATA>"; shows 'TypeDescription'
embedded screen at (762,3)-(888,87): SPRACHE_MENUE
3 more shapes without text or variables
*)

(* Visualisation ZLIB_ERRORLINE
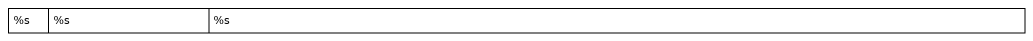
rectangle at (0,0)-(41,25): text "%s"; shows $ErrorStruct$.No; invisible if $ErrorStruct$.No = 0; dynamic style $ErrorStruct$.LineColor, $ErrorStruct$.LineColor
rectangle at (200,0)-(1017,25): text "%s"; shows $ErrorStruct$.Text; invisible if $ErrorStruct$.No = 0; dynamic style $ErrorStruct$.LineColor, $ErrorStruct$.LineColor
rectangle at (40,0)-(201,25): text "%s"; shows $ErrorStruct$.DateTime; invisible if $ErrorStruct$.No = 0; dynamic style $ErrorStruct$.LineColor, $ErrorStruct$.LineColor
*)

(* Visualisation ZLIB_ERRORLIST
